(* IEC 61131-3 sources: ZUT-informatyka/Semestr 5/PUA/Projekt Wiertarka, 3 files *)

(* ---- Types.typ ---- *)
TYPE
	StateMachineEnum: (
		INIT := 0, (* Drill waiting for start signal *)
		DRILL_PREP := 1, (* Drill preparation for work *)
		DRILLING := 2, (* Drilling in progress *)
		RETRACTING :=3, (* Drill retracting after drilling is done *)
		DRILL_STOPPING := 4, (* Drilling stopping *)
		PAUSED := 5, (* Drilling paused *)
		FAILURE := 6 (* Error occured *)
	);

	FailureEnum: (
		NO_ERROR := 0, (* No error *)
		DRILL_MOTOR_NOK := 1, (* Drill motor didn't turn on *)
		END_POS_UNREACHABLE := 2, (* Drill couldn't reach end position *)
		START_POS_UNREACHABLE := 3, (* Dril couldn't reach start position *)
		DRILL_MOTOR_OVERHEAT := 4, (* Drill motor overheated *)
		ESTOP := 5 (* EStop pressed *)
	);

	AlarmsStruct : STRUCT
		current : ARRAY[0..9] OF BOOL;
		acknowledge : ARRAY[0..9] OF BOOL;
	END_STRUCT;

	OperatorStruct : STRUCT
		diStart : BOOL; (* Start button *)
		diStop : BOOL;	(* Stop button *)
		diEStop : BOOL; (* Emergency stop button *)
		diConfirmFailure : BOOL; (* Failure clear button *)
		doActive : BOOL; (* Active state *)
	END_STRUCT;

	LightsStruct : STRUCT
		doActiveLED : BOOL; (* Machine active LED *)
		doPausedLED : BOOL; (* Machine paused LED *)
		doFailureLED : BOOL; (* Machine stopped because of error LED *)
	END_STRUCT;

	DrillStruct : STRUCT
		diThermMotorOK : BOOL; (* Motor temperature sensor *)
		diPowerMotorOK : BOOL; (* Motor power sensor *)
		doPowerMotor : BOOL; (* Drill motor power switch *)
		doDirMotor : BOOL; (* Drill direction switch; TRUE - clockwise, FALSE - counter clockwise *)
	END_STRUCT;

	FeedStruct : STRUCT
		diStartPosition : BOOL; (* Drill top position sensor *)
		diEndPosition : BOOL; (* Drill bottom position sensor *)
		doFeedPower : BOOL; (* Feeding motor power switch *)
		doDirFeed : BOOL; (* Drill vertical direction; TRUE - downwards, FALSE - upwards *)
	END_STRUCT;
END_TYPE

(* ---- Main.st ---- *)
PROGRAM _CYCLIC
	IF NOT(Operator.diEStop) THEN (* If Estop pressed, go to failure *)
		FailureReason := ESTOP;
		Alarms.current[0] := TRUE;
		StateMachine := FAILURE;
	END_IF;

	IF Drill.diThermMotorOK THEN (* If engine overheats, throw error *)
		FailureReason := DRILL_MOTOR_OVERHEAT;
		Alarms.current[1] := TRUE;
		StateMachine := FAILURE;
	END_IF;

	gAlarm := FALSE; (* Handling alarms *)
	FOR i := 0 TO 9 DO
		IF Alarms.current[i] OR Alarms.acknowledge[i] THEN
			gAlarm := TRUE;
		END_IF;
	END_FOR;

	CASE StateMachine OF
		INIT:
			CheckDrillEngineTON.IN := FALSE; (* Reset timers *)
			CheckDrillEngineTON();
			LiftingFeedTON.IN := FALSE;
			LiftingFeedTON();
			LoweringFeedTON.IN := FALSE;
			LoweringFeedTON();
			PauseDrillTON.IN := FALSE;
			PauseDrillTON();
			StopDrillTON.IN := FALSE;
			StopDrillTON();

			Operator.doActive := FALSE;
			ActivateSystemTON(IN := Operator.diStart, PT := T#2.0s); (* Wait for start button *)
			Operator.doActive := ActivateSystemTON.Q;

			IF Operator.doActive AND NOT(Drill.diThermMotorOK) THEN
				IF NOT(Feed.diStartPosition) THEN (* If feed not in start position, try to reach it *)
					Feed.doDirFeed := TRUE;
					Feed.doFeedPower := TRUE;

					LiftingFeedTON(IN := NOT(Feed.diStartPosition), PT := T#5.0s);

					IF LiftingFeedTON.Q THEN (* If start position unreachable, throw error *)
						FailureReason := START_POS_UNREACHABLE;
						Alarms.current[3] := TRUE;
						StateMachine := FAILURE;
					END_IF;
				END_IF;

				Lights.doActiveLED := TRUE; (* Activate active LED and go to drill preparation *)
				StateMachine := DRILL_PREP;
			END_IF;

		DRILL_PREP:
			Drill.doDirMotor := TRUE; (* Set drilling direction and power on the motor *)
			Drill.doPowerMotor := TRUE;

			CheckDrillEngineTON(IN := NOT(Drill.diPowerMotorOK), PT := T#5.0s); (* Limit time to turn on engine to 5s *)
			IF CheckDrillEngineTON.Q THEN (* If engine didn't turn on, throw error *)
				FailureReason := DRILL_MOTOR_NOK;
				Alarms.current[2] := TRUE;
				StateMachine := FAILURE;
			END_IF;

			IF Drill.diPowerMotorOK THEN (* If motor works start drilling *)
				StateMachine := DRILLING;
			END_IF;

		DRILLING:
			Feed.doDirFeed := TRUE; (* Set feed direction and power it *)
			Feed.doFeedPower := TRUE;

			LoweringFeedTON(IN := NOT(Feed.diEndPosition), PT := T#15.0s); (* Limit time to reach end position to 15s *)
			IF LoweringFeedTON.Q THEN (* If end position not reached, throw error *)
				FailureReason := END_POS_UNREACHABLE;
				Alarms.current[4] := TRUE;
				StateMachine := FAILURE;
			END_IF;

			PauseDrillTON(IN := Operator.diStop, PT := T#0.5s); (* Check if operator pauses or stops process *)
			StopDrillTON(IN := Operator.diStop, PT := T#2.0s);
			IF PauseDrillTON.Q THEN
				PauseHelperFlag := TRUE;
			END_IF;
			IF PauseHelperFlag AND NOT Operator.diStop THEN
				PauseHelperFlag := FALSE;
				StateMachine := PAUSED;
			END_IF;
			IF StopDrillTON.Q THEN
				StateMachine := DRILL_STOPPING;
			END_IF;

			IF Feed.diEndPosition THEN
				StateMachine := RETRACTING;	(* If drill reaches final position, start retracting *)
			END_IF;

		RETRACTING:
			Feed.doDirFeed := FALSE; (* Change feed and drill directions *)
			Drill.doDirMotor := FALSE;

			LiftingFeedTON(IN := NOT(Feed.diStartPosition), PT := T#5.0s); (* Limit time to retract to 5s *)
			IF LiftingFeedTON.Q THEN (* If start position not reached, throw error *)
				FailureReason := START_POS_UNREACHABLE;
				Alarms.current[3] := TRUE;
				StateMachine := FAILURE;
			END_IF;

			IF Feed.diStartPosition THEN
				Feed.doFeedPower := FALSE; (* If drill reaches start position, turn off feed and start drill stopping*)
				StateMachine := DRILL_STOPPING;
			END_IF;

		DRILL_STOPPING:
			Drill.doPowerMotor := FALSE; (* Turning off drill motor *)

			CheckDrillEngineTON(IN := Drill.diPowerMotorOK, PT := T#5.0s); (* Limit time to turn off engine to 5s *)
			IF CheckDrillEngineTON.Q THEN (* If engine didn't turn off, throw error *)
				FailureReason := DRILL_MOTOR_NOK;
				Alarms.current[2] := TRUE;
				StateMachine := FAILURE;
			END_IF;

			IF NOT(Drill.diPowerMotorOK) THEN
				StateMachine := INIT; (* If drill motor turns off, go to init state *)
			END_IF;

		PAUSED:
			Feed.doFeedPower := FALSE; (* Turn off feed and drill motor, turn on paused LED *)
			Drill.doPowerMotor := FALSE;

			CheckDrillEngineTON.IN := FALSE; (* Reset timers *)
			CheckDrillEngineTON();
			LiftingFeedTON.IN := FALSE;
			LiftingFeedTON();
			LoweringFeedTON.IN := FALSE;
			LoweringFeedTON();
			PauseDrillTON.IN := FALSE;
			PauseDrillTON();
			StopDrillTON.IN := FALSE;
			StopDrillTON();

			BlinkLedOnTON(IN := NOT(BlinkLedOffTON.Q), PT := T#1.0s);
			BlinkLedOffTON(IN := BlinkLedOnTON.Q, PT := T#1.0s);
			Lights.doPausedLED := BlinkLedOnTON.Q AND NOT(BlinkLedOffTON.Q);

			IF NOT(Drill.diPowerMotorOK) THEN (* If motor stopped, wait for start or abort *)
				IF EDGEPOS(Operator.diStart) THEN
					Lights.doPausedLED := FALSE; (* If start then resume drilling *)
					StateMachine := DRILLING;
				END_IF;

				IF EDGEPOS(Operator.diStop) THEN
					Feed.doFeedPower := TRUE; (* If stop then turn on feed and drill and start retracting *)
					Drill.doPowerMotor := TRUE;
					Lights.doPausedLED := FALSE;
					StateMachine := RETRACTING;
				END_IF;
			END_IF;

		FAILURE:
			CheckDrillEngineTON.IN := FALSE; (* Reset timers *)
			CheckDrillEngineTON();
			LiftingFeedTON.IN := FALSE;
			LiftingFeedTON();
			LoweringFeedTON.IN := FALSE;
			LoweringFeedTON();
			PauseDrillTON.IN := FALSE;
			PauseDrillTON();
			StopDrillTON.IN := FALSE;
			StopDrillTON();

			Feed.doFeedPower := FALSE; (* If failure occurs, turn off feed, drill and active led *)
			Drill.doPowerMotor := FALSE;
			Operator.doActive := FALSE;
			Lights.doActiveLED := FALSE;

			BlinkLedOnTON(IN := NOT(BlinkLedOffTON.Q), PT := T#1.0s);
			BlinkLedOffTON(IN := BlinkLedOnTON.Q, PT := T#1.0s);
			Lights.doFailureLED := BlinkLedOnTON.Q AND NOT(BlinkLedOffTON.Q);

			IF EDGEPOS(Operator.diConfirmFailure) AND NOT(Operator.diEStop) THEN (* If failure resolved, clear failure reason and go to init state *)
				Lights.doFailureLED := FALSE;
				FailureReason := NO_ERROR;
				FOR i := 0 TO 9 DO
					Alarms.current[i] := FALSE;
				END_FOR;
				StateMachine := INIT;
			END_IF;
	END_CASE;
END_PROGRAM

(* ---- Variables.var ---- *)
VAR
	(* Structures *)
	StateMachine : StateMachineEnum;
	FailureReason : FailureEnum;
	Operator : OperatorStruct;
	Lights : LightsStruct;
	Drill : DrillStruct;
	Feed : FeedStruct;

	(* Alarms *)
	Alarms : AlarmsStruct;
	gAlarm : BOOL;
	i : UINT;

	(* Timers *)
	ActivateSystemTON : TON; (* Checks start button for start input *)
	PauseDrillTON : TON; (* Checks stop button for pause input *)
	StopDrillTON : TON; (* Checks stop button for stop input *)
	CheckDrillEngineTON : TON; (* Checks if drill engine turns on *)
	LiftingFeedTON : TON; (* Checks if feed lifts *)
	LoweringFeedTON : TON; (* Checks if feeds lowers *)
	BlinkLedOnTON : TON; (* Timers to blink LEDs *)
	BlinkLedOffTON : TON;
	PauseHelperFlag : BOOL;
END_VAR
